TYPE ST_ManualAnalogAxisCtrl :
STRUCT
	bCmdRunCW	: BOOL ;
	bCmdRunCCW	: BOOL ;
	fCmdVelocity: LREAL ; 
	
END_STRUCT
END_TYPE

(* stored: Version 1.1.0.1, ProductVersion 3.1.4024.5
   DUT ST_ManualAnalogAxisCtrl: Id {a0675b15-8e0a-0e05-2d56-c1eb0c67c1b7} *)
